# EPICS StreamDevice protocol: catflwrSup/catflwr.proto
OutTerminator = "\r";
InTerminator = "\r";

ReplyTimeout = 2000;

get_st_array {
    in "%d,%d,%d"
}
